{attribute 'pack_mode' := '2'}
TYPE ST_XPU_CTRL :
STRUCT
  Cmd             : E_XPU_CTRL;
END_STRUCT
END_TYPE

(* stored: Version 1.1.0.1
   DUT ST_XPU_CTRL: Id {4551251e-da2e-4053-8c18-ccd1c2f9cd0b} *)
